TYPE ST_BaseHMITopElement_View :
STRUCT
	bDanaTopElement				: BOOL;
END_STRUCT
END_TYPE

(* stored: Version 1.1.0.1
   DUT ST_BaseHMITopElement_View: Id {b407ef35-511d-0539-2687-37f9a6583220} *)
